// TIA Portal V18 export
DATA_BLOCK "TD_Start_CAT_DB"   // DB14
// stored: AutoNumber false, InstanceOfName TD_Motor_Start_CAT, InstanceOfType FB
"TD_Motor_Start_CAT"
   // VAR
   //    EngineFault_TON { S7_SetPoint := 'True'} : TON_TIME;
   // END_VAR
BEGIN
END_DATA_BLOCK
